FUNCTION_BLOCK FB_GroupCA
VAR_IN_OUT
	ax					: ARRAY [1..Tc3_XTS_Utility.TcIoXtsEnvironmentParameterList.MaxXtsMoversPerXpu] OF fb_Mover;
END_VAR
VAR_INPUT
	fbXPUGroupCA		: FB_Mc2CaGroup;
END_VAR
VAR_OUTPUT
	eGroupState			: MC_GROUP_STATE;
	bAllStandStill		: BOOL;
	bError				: BOOL;
END_VAR
VAR 
	//Function Blocks
	ag					: AXES_GROUP_REF;
	fbEnable			: MC_GroupEnable;
	fbDisable			: MC_GroupDisable;
	fbHalt				: MC_GroupHalt;
	fbUnGroupAll		: MC_UngroupAllAxes;
	fbGroupStop			: MC_GroupStop;
	fbReset				: MC_GroupReset;
	fbState				: MC_GroupReadStatus;
END_VAR

fbEnable(
	AxesGroup:= ag, 
	Execute:= , 
	Done=> , 
	Busy=> , 
	Error=> , 
	ErrorId=> );
	
fbDisable(
	AxesGroup:= ag, 
	Execute:= , 
	Done=> , 
	Busy=> , 
	Error=> , 
	ErrorId=> );
	
fbGroupStop(
	AxesGroup:= ag, 
	Execute:= , 
	Deceleration:= , 
	Jerk:= , 
	Done=> , 
	Busy=> , 
	Active=> , 
	CommandAborted=> , 
	Error=> , 
	ErrorId=> );
	
fbHalt(
	AxesGroup:= ag, 
	Execute:= , 
	Deceleration:= , 
	Jerk:= , 
	Done=> , 
	Busy=> , 
	Active=> , 
	CommandAborted=> , 
	Error=> , 
	ErrorId=> );
	
fbUnGroupAll(
	AxesGroup:= ag, 
	Execute:= , 
	Done=> , 
	Busy=> , 
	Error=> , 
	ErrorId=> );
	
fbReset(
	AxesGroup:= ag, 
	Execute:= , 
	Done=> , 
	Busy=> , 
	Error=> , 
	ErrorId=> );
	
fbState(
	AxesGroup:= ag, 
	Enable:= TRUE, 
	Valid=> , 
	Busy=> , 
	GroupMoving=> , 
	GroupHoming=> , 
	GroupErrorStop=> , 
	GroupNotReady=> , 
	GroupStandby=> , 
	GroupStopping=> , 
	GroupDisabled=> , 
	AllAxesStanding=> , 
	ConstantVelocity=> , 
	Accelerating=> , 
	Decelerating=> , 
	InPosition=> , 
	Error=> , 
	ErrorId=> );
	
IF fbState.GroupDisabled THEN
	eGroupState := MC_GROUP_STATE.mcGroupStateDisabled;
ELSIF fbState.GroupErrorStop THEN
	eGroupState := MC_GROUP_STATE.mcGroupStateErrorStop;
ELSIF fbState.GroupHoming THEN
	eGroupState := MC_GROUP_STATE.mcGroupStateHoming;
ELSIF fbState.GroupMoving THEN
	eGroupState := MC_GROUP_STATE.mcGroupStateMoving;
ELSIF fbState.GroupNotReady THEN
	eGroupState := MC_GROUP_STATE.mcGroupStateNotReady;
ELSIF fbState.GroupStandby THEN
	eGroupState := MC_GROUP_STATE.mcGroupStateStandby;
ELSIF fbState.GroupStopping THEN
	eGroupState := MC_GROUP_STATE.mcGroupStateStopping;
ELSIF fbState.GroupStandby THEN
	eGroupState := MC_GROUP_STATE.mcGroupStateSuspended;
ELSE
	eGroupState := MC_GROUP_STATE.mcGroupStateInvalid;
END_IF
bError := eGroupState = mc_group_state.mcGroupStateErrorStop;
bAllStandStill := fbState.AllAxesStanding;

METHOD m_clearCmd : BOOL
VAR_INPUT
END_VAR
m_halt(FALSE);
m_reset(FALSE);
m_ungroupall(FALSE);
m_enable(FALSE);
m_disable(FALSE);
END_METHOD

METHOD m_disable : bool
VAR_INPUT
	bExecute : BOOL;
END_VAR
fbDisable.Execute 	:= bExecute;
m_disable			:= fbDisable.Done;
END_METHOD

METHOD m_enable : bool
VAR_INPUT
	bEnable : BOOL;
END_VAR
fbEnable.Execute 	:= bEnable;
m_enable			:= fbEnable.Done;
END_METHOD

METHOD m_halt : bool
VAR_INPUT
	bExecute : BOOL;
END_VAR
fbHalt.Execute 		:= bExecute;
m_halt				:= fbHalt.Done;
END_METHOD

METHOD m_reset : bool
VAR_INPUT
	bREset : BOOL;
END_VAR
fbReset.Execute := bREset;
m_reset			:= fbReset.Done;
END_METHOD

METHOD m_ungroupall : bool
VAR_INPUT
	bExecute :BOOL;
END_VAR
fbUnGroupAll.Execute 	:= bExecute;
m_ungroupall			:= fbUnGroupAll.Done;
END_METHOD

END_FUNCTION_BLOCK

(* stored: Version 1.1.0.1, ProductVersion 3.1.4024.11
   POU FB_GroupCA: Id {6e35faa1-0ee4-41ef-8125-56a7113871cf}, SpecialFunc None
   Method m_clearCmd: Id {bd3f94be-b975-4f0a-abfd-bd17a7fb4a02}
   Method m_disable: Id {7ed6aefe-997e-4a60-9014-c0c3ac681d26}
   Method m_enable: Id {68e53748-7c17-4773-81e7-db15626d6f4a}
   Method m_halt: Id {370dfd46-8ee9-4be6-a974-a26aacf35016}
   Method m_reset: Id {d117629c-f8ec-4af1-aeb9-7b88477d6bb0}
   Method m_ungroupall: Id {c4d04756-20dc-4d04-9707-7855a191fb37} *)
